FUNCTION_BLOCK GET_XY_COORD (* Set a destination point with a 'z' axis constant *)
  (* Standard: 61499-2 *)
  (* Version 1.0, 09-01-12, GASR, Universidade do Estado de Santa Catarina *)
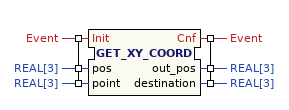
  EVENT_INPUT
    Init WITH pos, point; (* Initialization request *)
  END_EVENT
  EVENT_OUTPUT
    Cnf WITH out_pos, destination; (* Execution confirmed *)
  END_EVENT
  VAR_INPUT
    pos : ARRAY [0..2] OF REAL; (* Machine position *)
    point : ARRAY [0..2] OF REAL; (* Point with X and Y coordinates *)
  END_VAR
  VAR_OUTPUT
    out_pos : ARRAY [0..2] OF REAL; (* Machine position *)
    destination : ARRAY [0..2] OF REAL; (* Point with z axis constant *)
  END_VAR
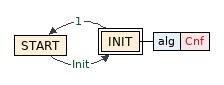
  EC_STATES
    INIT : alg -> Cnf;
    START;
  END_STATES
  EC_TRANSITIONS
    START TO INIT := Init;
    INIT TO START := 1;
  END_TRANSITIONS
  ALGORITHM alg IN Lua:
 local i for i = 1, 3 do  out_pos[ i ] = pos[ i ] end destination[ 1 ] = point[ 1 ] destination[ 2 ] = point[ 2 ] destination[ 3 ] = pos[ 3 ]
  END_ALGORITHM
END_FUNCTION_BLOCK
